TYPE EleControlNo ://气缸、真空阀、破真空阀
STRUCT
	CylinderName:ST_CylinderName;//气缸号
	ElectValveName:ST_ElectValveName;//真空和破真空号
END_STRUCT
END_TYPE

(* stored: Version 1.1.0.1, ProductVersion 3.1.4024.9
   DUT EleControlNo: Id {dab86100-ff8e-43de-985f-165701a4a037} *)
